// TwinCAT 3 PLC project RT1
// ProgramVersion: 3.1.4023.0
// libraries:
//   Tc2_ModbusRTU, * (Beckhoff Automation GmbH)
//   Tc2_Standard, * (Beckhoff Automation GmbH)
//   Tc2_System, * (Beckhoff Automation GmbH)
//   Tc2_Utilities, * (Beckhoff Automation GmbH)
//   Tc3_Module, * (Beckhoff Automation GmbH)
// project tree:
//   DUTs/ E_ROOM_TEMP_STS.TcDUT, ST_ROOM.TcDUT
//   GVLs/ GVL.TcGVL
//   / PlcTask.TcTTO
//   POUs/ FB_Motor.TcPOU, F_AnalogScale.TcPOU, MAIN.TcPOU, prgLab02.TcPOU, prgLab04_06.TcPOU, prgLab05_07.TcPOU, prgLab08.TcPOU, prgLab10_11.TcPOU, prgLab14B.TcPOU, prgLab16.TcPOU, prgLab3A.TcPOU, P_Divisao.TcPOU
// real-time tasks:
//   TASK PlcTask: cycle T#10ms, priority 20, ADS port 350
// motion (NC):
//   TASK NC-Task 1 SAF: cycle T#2ms, priority 4, ADS port 501
//   TASK NC-Task 1 SVB: cycle T#10ms, priority 8, ADS port 511
//   AXIS Axis 1 (id 1)
// I/O:
//   DEVICE Device 3 (EtherCAT) (disabled), AmsNetId 192.168.0.60.4.1
//     Term 1 (EK1100) [EK1100 EtherCAT Coupler (2A E-Bus)]
//       Term 2 (EL1012) [EL1012 2Ch. Dig. Input 24V, 10µs]
//       Term 3 (EL1012)
//       Term 4 (EL1012) [EL1012 2Ch. Dig. Input 24V, 10µs]
//       Term 5 (EL1012)
//       Term 6 (EL2004)
//       Term 7 (EL4002) [EL4002 2Ch. Ana. Output 0-10V, 12bit]
//       Term 8 (EL9512) [EL9512 Power supply terminal 12V]
//       Term 9 (EL3102)
//       Term 10 (EL9011)
// variable links:
//   RT1 Instance <-> Device 3 (EtherCAT)/Term 1 (EK1100)/Term 2 (EL1012)
//     PlcTask Inputs/prgLab14B.b1 <-> Channel 1/Input

CONFIGURATION RT1
    RESOURCE PLC ON TwinCAT3
        TASK PlcTask(INTERVAL := T#10ms, PRIORITY := 20);
        PROGRAM MAIN WITH PlcTask : MAIN;
    END_RESOURCE
END_CONFIGURATION

// ---- DUTs/E_ROOM_TEMP_STS.TcDUT
{attribute 'qualified_only'}
{attribute 'strict'}
TYPE E_ROOM_TEMP_STS :
(
	baixa:=1,
	normal:=2,
	moderada:=3,
	alta:=4,
	muito_alta:=5
);
END_TYPE

// ---- DUTs/ST_ROOM.TcDUT
TYPE ST_ROOM :
STRUCT
	OccupancySensor: BOOL;	//Sensor de ocupação
	Lighting:BOOL;          //Iluminação
	Heating:BOOL;           //Aquecimento
	Ventilation:BOOL;       //Ventilador
	AirQuality: REAL;       //Qualidade do ar
	setpoint:REAL:=50;      //Setpoint
	Temp:REAL;
	status:E_ROOM_TEMP_STS;
END_STRUCT
END_TYPE

// ---- GVLs/GVL.TcGVL
{attribute 'qualified_only'}
VAR_GLOBAL
	Room1:ST_ROOM;
	statusRoom1:E_ROOM_TEMP_STS;
	aRooms:ARRAY[1..3] OF ST_ROOM;
END_VAR
VAR_GLOBAL PERSISTENT
	iPersistent:INT;
	sPersistent:STRING;
	rPersistent:REAL;
END_VAR

// ---- POUs/MAIN.TcPOU
PROGRAM MAIN
VAR
	
END_VAR

prgLab02();
prgLab3A();
prgLab04_06();
prgLab05_07();
prgLab08();
prgLab14B();
prgLab10_11();
prgLab16();

END_PROGRAM

// ---- POUs/prgLab02.TcPOU
PROGRAM prgLab02
VAR
	contadorUp:CTU;
	contUp: BOOL;
	resetCount: BOOL;
	countFinished: BOOL;
	counterV: WORD;
	
	trig:R_TRIG;
	bTrigCnt:BOOL;
	contagemAtual:UDINT;
	
	passoContagem: UDINT:=1;
	fimContagem: BOOL;

	contagemProgramada: UDINT:=5;
	
	di1 AT %I*:BOOL;
	do1 AT %Q*:BOOL;
	do2 AT %Q*:BOOL;
	entradaAnalogica AT %I*:INT;
END_VAR
VAR CONSTANT
	var5Volts :INT:=16383;	//32767/2
END_VAR

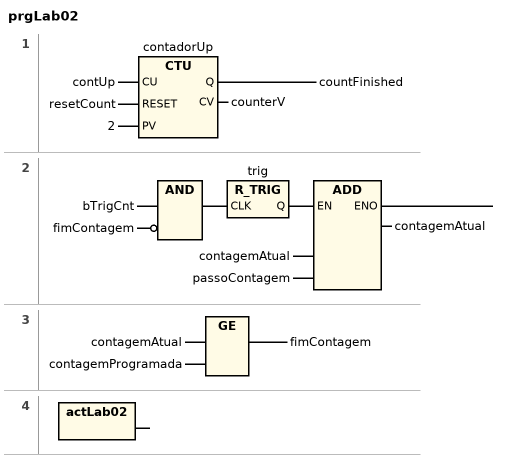
// NETWORK 1
contadorUp(CU := contUp, RESET := resetCount, PV := 2, CV => counterV); // CTU
countFinished := contadorUp.Q;

// NETWORK 2
trig(CLK := bTrigCnt AND NOT fimContagem); // R_TRIG
IF trig.Q THEN contagemAtual := contagemAtual + passoContagem; END_IF

// NETWORK 3
fimContagem := contagemAtual >= contagemProgramada;

// NETWORK 4
actLab02();

ACTION actLab02:
IF di1 THEN
	do1 := entradaAnalogica>= var5Volts;
	do2:= NOT do1;
ELSIF NOT di1 THEN
	do2 := entradaAnalogica>= var5Volts;
	do1:= NOT do2;		
END_IF
END_ACTION

END_PROGRAM

// ---- POUs/prgLab3A.TcPOU
PROGRAM prgLab3A
VAR
	aInteiros:ARRAY[0..8] OF INT;
	aBools:ARRAY[0..8] OF BOOL;
	
	i: INT;
	ai:ARRAY[1..5] OF INT;
END_VAR

FOR i:=0 TO 8 DO
	aBools[i]:= aInteiros[i]>10;
END_FOR

FOR i:=1 TO 5 DO
	ai[i]:=i;
END_FOR

END_PROGRAM

// ---- POUs/prgLab04_06.TcPOU
PROGRAM prgLab04_06
VAR
END_VAR

//Primeiro iremos conduzir as comparações básicas

IF GVL.Room1.OccupancySensor THEN
	GVL.Room1.Lighting:=TRUE;
	IF GVL.Room1.Temp > 24 THEN
		GVL.Room1.Heating:=FALSE;
	ELSIF GVL.Room1.Temp <20 THEN
		GVL.Room1.Heating:=TRUE;	
	END_IF
ELSE
	GVL.Room1.Lighting:=GVL.Room1.Heating:=FALSE;	
END_IF
IF GVL.Room1.AirQuality >= GVL.Room1.setpoint THEN
	GVL.Room1.Ventilation:=TRUE;
ELSE
	GVL.Room1.Ventilation:=FALSE;	
END_IF
//Solução lab 06
IF GVL.Room1.Temp< 20 THEN
	GVL.statusRoom1:= E_ROOM_TEMP_STS.baixa;
ELSIF GVL.Room1.Temp >=20 AND GVL.Room1.Temp < 24 THEN
	GVL.statusRoom1:= E_ROOM_TEMP_STS.normal;
ELSIF GVL.Room1.Temp >=24 AND GVL.Room1.Temp < 27 THEN
	GVL.statusRoom1:= E_ROOM_TEMP_STS.moderada;
ELSIF GVL.Room1.Temp >=27 AND GVL.Room1.Temp < 32 THEN
	GVL.statusRoom1:= E_ROOM_TEMP_STS.alta;
ELSIF GVL.Room1.Temp >=32 THEN
	GVL.statusRoom1:= E_ROOM_TEMP_STS.muito_alta;
END_IF

END_PROGRAM

// ---- POUs/prgLab05_07.TcPOU
PROGRAM prgLab05_07
VAR
	i: INT;
END_VAR

//Na segunda parte desse mesmo exercício o objetivo é basicamente de expandí-lo transformando o que era um único
//Elemento em um vetor de 3

FOR i:=1 TO 3 DO
	IF GVL.aRooms[i].OccupancySensor THEN
		GVL.aRooms[i].Lighting:=TRUE;
		IF GVL.aRooms[i].Temp > 24 THEN
			GVL.aRooms[i].Heating:=FALSE;
		ELSIF GVL.aRooms[i].Temp <20 THEN
			GVL.aRooms[i].Heating:=TRUE;	
		END_IF
	ELSE
		GVL.aRooms[i].Lighting:=GVL.aRooms[i].Heating:=FALSE;	
	END_IF
	IF GVL.aRooms[i].AirQuality >= GVL.aRooms[i].setpoint THEN
		GVL.aRooms[i].Ventilation:=TRUE;
	ELSE
		GVL.aRooms[i].Ventilation:=FALSE;	
	END_IF	
	//Solução Lab 07
	IF GVL.aRooms[i].Temp< 20 THEN
		GVL.aRooms[i].status:= E_ROOM_TEMP_STS.baixa;
	ELSIF GVL.aRooms[i].Temp >=20 AND GVL.aRooms[i].Temp < 24 THEN
		GVL.aRooms[i].status:= E_ROOM_TEMP_STS.normal;
	ELSIF GVL.aRooms[i].Temp >=24 AND GVL.aRooms[i].Temp < 27 THEN
		GVL.aRooms[i].status:= E_ROOM_TEMP_STS.moderada;
	ELSIF GVL.aRooms[i].Temp >=27 AND GVL.aRooms[i].Temp < 32 THEN
		GVL.aRooms[i].status:= E_ROOM_TEMP_STS.alta;
	ELSIF GVL.aRooms[i].Temp >=32 THEN
		GVL.aRooms[i].status:= E_ROOM_TEMP_STS.muito_alta;
	END_IF	
END_FOR

END_PROGRAM

// ---- POUs/prgLab08.TcPOU
PROGRAM prgLab08
VAR
	writePersistent:FB_WritePersistentData;
	error: BOOL;
	start: BOOL;
END_VAR
VAR PERSISTENT
	iPersistLocal:INT;
END_VAR

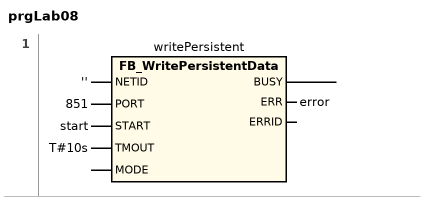
// NETWORK 1
writePersistent(NETID := '', PORT := 851, START := start, TMOUT := T#10s, ERR => error); // FB_WritePersistentData

END_PROGRAM

// ---- POUs/prgLab14B.TcPOU
PROGRAM prgLab14B
VAR
	r1:REAL:=10;
	r2:REAL:=1;
	r3:REAL;
	b1 AT %I*:BOOL;
END_VAR

IF b1 THEN
	r2:=0;
END_IF

r3:=r1/r2;

END_PROGRAM

// ---- POUs/prgLab10_11.TcPOU
PROGRAM prgLab10_11
VAR
	motor:FB_Motor;
	bLiga AT %I*: BOOL;
	bDesliga AT %I*: BOOL;
	reset AT %I*: BOOL;
	temperatura: REAL;
	saidaMotor AT %Q*: BOOL;
	error AT %Q*: BOOL;
	analogInput AT %I*: INT;
END_VAR

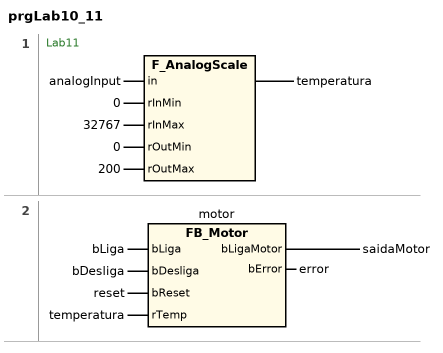
// NETWORK 1
// Lab11
temperatura := F_AnalogScale(in := analogInput, rInMin := 0, rInMax := 32767, rOutMin := 0, rOutMax := 200);

// NETWORK 2
motor(bLiga := bLiga, bDesliga := bDesliga, bReset := reset, rTemp := temperatura, bError => error); // FB_Motor
saidaMotor := motor.bLigaMotor;

END_PROGRAM

// ---- POUs/FB_Motor.TcPOU
FUNCTION_BLOCK FB_Motor
VAR_INPUT
	bLiga, bDesliga, bReset:BOOL;
	rTemp:REAL;
END_VAR
VAR_OUTPUT
	bLigaMotor, bError:BOOL;
END_VAR
VAR
END_VAR

IF rTemp >=100 THEN
	bError:=TRUE;
END_IF
IF bLiga AND NOT bDesliga AND NOT bError AND rTemp<80 THEN
	bLigaMotor:=TRUE;
ELSIF bDesliga OR bError THEN
	bLigaMotor:=FALSE;
END_IF

IF bReset AND rTemp < 80 THEN
	bError:=FALSE;
END_IF

END_FUNCTION_BLOCK

// ---- POUs/F_AnalogScale.TcPOU
FUNCTION F_AnalogScale : REAL
VAR_INPUT
	in:INT;
	rInMin:REAL:=0;
	rInMax:REAL:=32767;
	rOutMin:REAL:=0;
	rOutMax:REAL:=200;
END_VAR
VAR
	
	validParams: BOOL;
END_VAR

validParams:= (rInMax-rInMin)>0;
IF validParams THEN
	F_AnalogScale:= INT_TO_REAL(in)*(rOutMax-rOutMin)/(rInMax-rInMin) + rOutMin;
END_IF

END_FUNCTION

// ---- POUs/prgLab16.TcPOU
PROGRAM prgLab16
VAR
	rAddSin:LREAL:=0.01;
	rResultSin:LREAL;
	rSin:LREAL;
	rAddTri:LREAL:=0.01;
	rResultTri:LREAL:=0.01;
	rTri:LREAL;
	rVector:ARRAY[1..5] OF LREAL:=[1,5,6,2,8];
END_VAR

rResultSin:=rResultSin+rAddSin;
rSin:=SIN(rResultSin);

rTri:=rTri+rResultTri;
IF rTri>=1 THEN
	rResultTri:= -rAddTri;
ELSIF rTri <=-1 THEN
	rResultTri:= rAddTri;
END_IF

END_PROGRAM

// ---- POUs/P_Divisao.TcPOU
PROGRAM P_Divisao
VAR
	bCalcular	: BOOL;
	rValor1		: REAL;
	rValor2		: REAL;
	rResultado	: REAL;
END_VAR

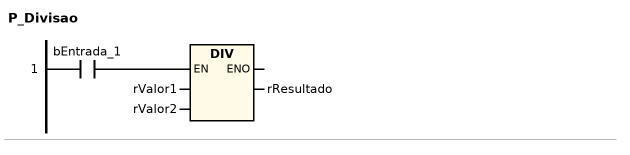
// NETWORK 1
IF bEntrada_1 THEN rResultado := rValor1 / rValor2; END_IF

END_PROGRAM
